// TIA Portal V20 export
DATA_BLOCK "DB_Temporary"   // DB40
// stored: MemoryReserve 100, Namespace EmptyLine
   VAR
      MABS1_In { ExternalAccessible := 'False'; ExternalVisible := 'False'; ExternalWritable := 'False'} : "Global.IB_P01_02_03_in_64bytes_struct";
      MABS1_Out { ExternalAccessible := 'False'; ExternalVisible := 'False'; ExternalWritable := 'False'} : "Global.IB_P01_02_03_out_64bytes_struct";
      MABS2_In { ExternalAccessible := 'False'; ExternalVisible := 'False'; ExternalWritable := 'False'} : "Global.IB_P01_02_03_in_64bytes_struct";
      MABS2_Out { ExternalAccessible := 'False'; ExternalVisible := 'False'; ExternalWritable := 'False'} : "Global.IB_P01_02_03_out_64bytes_struct";
   END_VAR
BEGIN
END_DATA_BLOCK
